Universal Robots PolyScope program: Change Spool.urp

Program Change Spool (installation=robot3 directory=/programs/UPF createdIn=5.14.5 lastSavedIn=5.21.2 robotSerialNumber=20256802612)
Calibrated DH parameters: a=[-0.000042, -0.384711, -0.675257, 0.000053, -0.000026, 0]; d=[0.236319, 419.71573, -259.410189, -160.105167, 0.159217, 0.154051]; alpha=[1.570689, 0.001837, -0.001695, 1.571673, -1.570506, 0]; deltaTheta=[0, 1.107921, -1.49058, 0.382655, 0.000001, 0]
InitVariablesNode
BeforeStart
  Folder premove
    Set NoAction tcp=pretend_welder
    cur_pos := get_actual_tcp_pose()
    MoveJ speed 60 deg/s, acceleration 80 deg/s^2 (useActiveTCP=true optimoveEnabled=false optiMoveSpeed=0.3 optiMoveAcceleration=0.09) feature=Base
      Waypoint Variable (Variable): variable=cur_pos
Robot Program (runOnlyOnce=false)
  'move robot above bucket'
  Set NoAction tcp=pretend_welder
  MoveJ speed 60 deg/s, acceleration 80 deg/s^2 (useActiveTCP=true optimoveEnabled=false optiMoveSpeed=0.3 optiMoveAcceleration=0.09) feature=Base
    Waypoint Waypoint_1: TCP in base x=454.836 y=405.454 z=142.442 mm, rx=2.3168 ry=2.0514 rz=0.0766 rad; joints [-187.619, -95.37, 137.796, -10.373, -0.811, -35.911] deg; TCP offset x=-5.49 y=-328 z=106.39 mm, rx=1.2092 ry=-1.2092 rz=1.2092 rad
  SuppressedNode
    URCap WireTank Serial (WireTank Serial, WireTank, LLC) dataModel(Command=[252,72,49], byte_array=true, NODE_TITLE=Serial Bridge uH1, QUERY=false, OUTPUT_ENTRY=Static, Variable(key=OUTPUT_VARIABLE, variable(name=HwResp)))
  Set DigitalOutput pin=digital_out[0]; digitalValue=1
  URCap WireTank Serial (WireTank Serial, WireTank, LLC) dataModel(NODE_TITLE=Serial Bridge uR1, Command=[252,82,49], QUERY=false, OUTPUT_ENTRY=Static, byte_array=true, Variable(key=OUTPUT_VARIABLE, variable=HwResp))
  SuppressedNode
    Script: popup(HwResp)
  SuppressedNode
    Wait Sleep waitTime=5
  Popup Message (haltProgram=false message=on inputType=Text)
  Set DigitalOutput pin=digital_out[0]; digitalValue=0
  URCap WireTank Serial (WireTank Serial, WireTank, LLC) dataModel(NODE_TITLE=Serial Bridge uR0, Command=[252,82,48], OUTPUT_ENTRY=Static, byte_array=true, QUERY=false, Variable(key=OUTPUT_VARIABLE, variable=HwResp))
  SuppressedNode
    Script: popup(HwResp)
  Popup Message (haltProgram=false message=off inputType=Text)
